
TYPE "TestAllTypes_001"
STRUCT
        CONFIG : "Config_001";
        STATUS : "Status_001";
        PROCESS_DATA : "ProcessData_001";
        MATRIX : "Matrix_001";
        ALARM_CONFIG : "AlarmConfig_001";
        ALARM_HISTORY : ARRAY[0..9] OF "Status_001";
        GRID : ARRAY[0..3,0..3] OF "ProcessData_001";
END_STRUCT;
END_TYPE